{attribute 'qualified_only'}
{attribute 'strict'}
TYPE TestEnum :
(
	first := 0,
	second := 1,
	third := 2
);
END_TYPE

(* stored: Version 1.1.0.1, ProductVersion 3.1.4024.9
   DUT TestEnum: Id {cc621b9e-fd25-4cd7-8df0-4a20201c2fa3} *)
